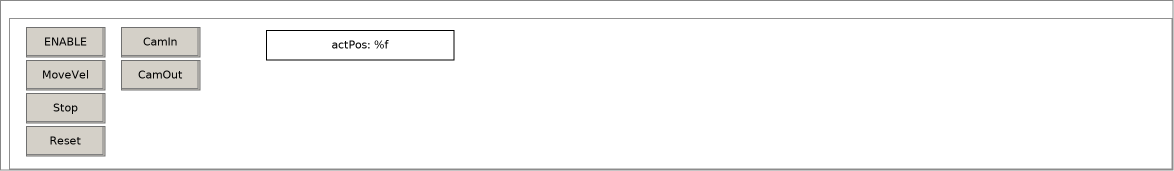
VISUALIZATION Vis_Axisadmin  // 1174x171
VAR_IN_OUT
	Axis: UDT_axisAdmin;
END_VAR
    GroupBox (9,10 1163x159)
        Button (17,17 79x30), "ENABLE"
            toggle Axis.i.Enable
        Button (17,50 79x30), "MoveVel"
            tap Axis.i.MoveVel
        Button (112,17 79x30), "CamIn"
            tap Axis.i.CamIn
        Button (112,50 79x30), "CamOut"
            tap Axis.i.CamOut
        Button (17,83 79x30), "Stop"
            tap Axis.i.Stop
        Button (17,116 79x30), "Reset"
            tap Axis.i.Reset
        RoundedRectangle (257,20 188x30), "actPos: %f", text variable: Axis.o.ActPos
END_VISUALIZATION

(* stored: Version 1.1.0.1, ProductVersion 3.1.4022.16
   Visu Vis_Axisadmin: Id {5a1ff5a1-8830-4a47-bb3a-8eb739b0f48b} *)
